FUNCTION_BLOCK differential_protection_1_2_backup2 (* Composite Function Block Type *)
  (* Standard: 61499-2 *)
  (* Version 0.0, 3/23/2016, gulzha, nxtControl GmbH, template *)
  PACKAGE Main;
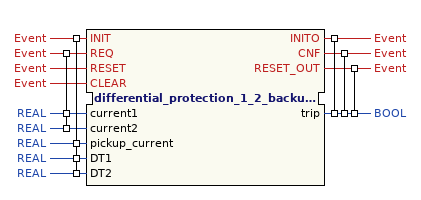
  EVENT_INPUT
    INIT WITH DT1, DT2, pickup_current; (* Initialization Request *)
    REQ WITH current1, current2; (* Normal Execution Request *)
    RESET;
    CLEAR;
  END_EVENT
  EVENT_OUTPUT
    INITO WITH trip; (* Initialization Confirm *)
    CNF WITH trip; (* Execution Confirmation *)
    RESET_OUT WITH trip;
  END_EVENT
  VAR_INPUT
    current1 : REAL;
    current2 : REAL;
    pickup_current : REAL;
    DT1 : REAL; (* Delay Time in seconds *)
    DT2 : REAL; (* Delay Time in seconds *)
  END_VAR
  VAR_OUTPUT
    trip : BOOL;
  END_VAR
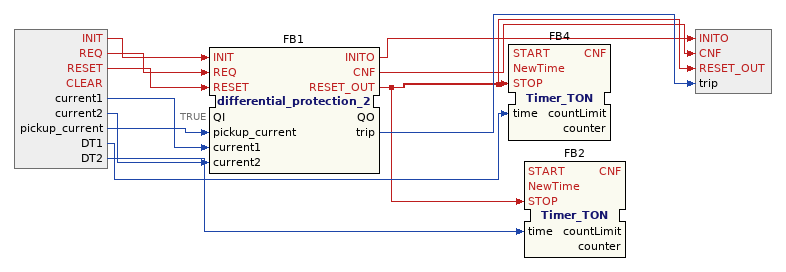
  FBS
    FB1 : differential_protection_2(QI := TRUE);
    FB4 : Timer_TON;
    FB2 : Timer_TON;
  END_FBS
  EVENT_CONNECTIONS
    INIT TO FB1.INIT;
    FB1.INITO TO INITO;
    FB1.CNF TO CNF;
    REQ TO FB1.REQ;
    RESET TO FB1.RESET;
    FB1.RESET_OUT TO FB4.STOP;
    FB1.RESET_OUT TO FB2.STOP;
    FB1.RESET_OUT TO RESET_OUT;
  END_CONNECTIONS
  DATA_CONNECTIONS
    FB1.trip TO trip;
    pickup_current TO FB1.pickup_current;
    current1 TO FB1.current1;
    current2 TO FB1.current2;
    DT1 TO FB4.time;
    DT2 TO FB2.time;
  END_CONNECTIONS
END_FUNCTION_BLOCK
